// TIA Portal V16 export
// export: Created 2022-11-24T15:20:45.6497294Z, ExportSetting WithDefaults, DisplayName Totally Integrated Automation Portal, DisplayVersion V16 Update 6, DisplayName TIA Portal Version Control Interface, DisplayVersion V16 Update 2, DisplayName TIA Portal Openness, DisplayVersion V16 Update 6, DisplayName SINAMICS Startdrive Advanced, DisplayVersion V16 Update 5, DisplayName SINAMICS Startdrive G130, G150, S120, S150, SINAMICS MV, S210, DisplayVersion V16 Update 5, DisplayName SINAMICS Startdrive G110M, G120, G120C, G120D, G120P, G115D, DisplayVersion V16 Update 5, DisplayName STEP 7 Professional, DisplayVersion V16 Update 6, DisplayName STEP 7 Safety, DisplayVersion V16, DisplayName WinCC Advanced, DisplayVersion V16 Update 6
FUNCTION "FC09_NoPressurePlate" : Void   // FC9, LAD
TITLE = Pressure palte isn't present
{ S7_Optimized_Access := 'FALSE' }
AUTHOR : Robopac
VERSION : 0.0
// stored: AutoNumber false, IsIECCheckEnabled false, SetENOAutomatically false, UDAEnableTagReadback false
BEGIN

REGION Network 1: Pressure plate bits
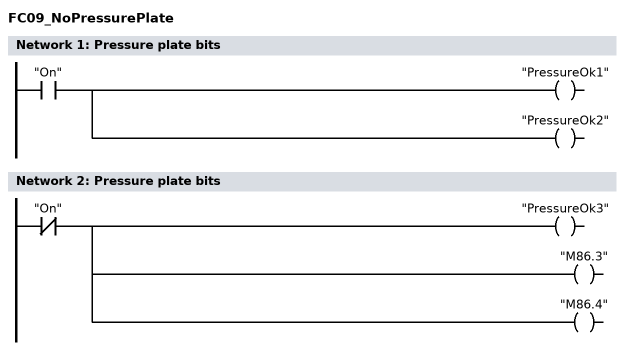
   RUNG wire#powerrail
      Contact( "On" )
      wire#w1
      Coil( "PressureOk1" )
   END_RUNG
   RUNG wire#w1
      Coil( "PressureOk2" )
   END_RUNG
   // the same network as SCL:
   "PressureOk1" := "On";
   "PressureOk2" := "On";
END_REGION

REGION Network 2: Pressure plate bits
   RUNG wire#powerrail
      I_Contact( "On" )
      wire#w1
      Coil( "PressureOk3" )
   END_RUNG
   RUNG wire#w1
      Coil( "M86.3" )
   END_RUNG
   RUNG wire#w1
      Coil( "M86.4" )
   END_RUNG
   // the same network as SCL:
   "PressureOk3" := NOT "On";
   "M86.3" := NOT "On";
   "M86.4" := NOT "On";
END_REGION
END_FUNCTION
